TYPE ST_GranSts :
STRUCT
    // Odwadnianie – 1=praca, 0=awaria/zanik
    bDewaterRun    : BOOL;

    // Silosy min
    bS01_Min       : BOOL;
    bS02_Min       : BOOL;

    // Klapa krańcówki / potwierdzenia
    bFlapOpen      : BOOL;
    bFlapClosed    : BOOL;
    bFlapInPos     : BOOL;    // jeśli masz (opcjonalnie)

    // Faulty napędów (z Twoich FB)
    bFault_SP02    : BOOL;
    bFault_SC01    : BOOL;
    bFault_SC02    : BOOL;
    bFault_M01     : BOOL;
    bFault_M02     : BOOL;
    bFault_Flap    : BOOL;

    // Waga (kg)
    rMassRawKg     : REAL;
END_STRUCT
END_TYPE

(* stored: Version 1.1.0.1, ProductVersion 3.1.4024.15
   DUT ST_GranSts: Id {31de6f5d-def5-460f-96a9-3a4304ca71c5} *)
